TYPE LG_get :
STRUCT
	Coils	:	LG_Coils;
	Status	:	LG_StatusBits;
	Data	:	LG_InputRegs;
	Control	:	LG_ControlRegs;	
END_STRUCT
END_TYPE

(* stored: Version 1.1.0.1, ProductVersion 3.1.4024.12
   DUT LG_get: Id {b63f487c-7d43-4145-ae34-7685c6ab7bdd} *)
